Yaskawa INFORM job: R1_W24(-90,90)KM-OK.JBI

/JOB
//NAME R1_W24(-90,90)KM-OK
///FOLDERNAME SCIANA-NOWY-R2-KM
//POS
///NPOS 55,55,0,5,0,0
///TOOL 0
///POSTYPE PULSE
///PULSE
C00000=-125210,-84514,-96282,42678,80589,-84145
C00001=-120727,25071,-5570,41830,73546,-76217
C00002=-120731,25851,-8598,41444,75264,-75512
C00003=-122137,52036,20168,42709,72709,-77203
C00004=-120675,58589,29768,42747,70121,-77648
C00005=-120167,58596,29776,42572,69880,-77517
C00006=-120675,58589,29768,42747,70121,-77648
C00007=-120675,58540,30899,42917,69583,-77884
C00008=-120675,58589,29768,42747,70121,-77648
C00009=-120675,58477,29643,42742,70137,-77641
C00010=-122267,58661,28071,43051,71685,-77708
C00011=-120675,58477,29643,42742,70137,-77641
C00012=-120223,58483,29649,42586,69921,-77523
C00013=-120675,58477,29643,42742,70137,-77641
C00014=-120675,58430,30663,42897,69653,-77855
C00015=-120675,58477,29643,42742,70137,-77641
C00016=-127422,61486,21154,43844,78340,-77144
C00017=-103662,71226,20496,-9632,86815,-77299
C00018=-86138,65266,24877,-44765,91557,-78354
C00019=-89288,46121,11206,-46267,89248,-79163
C00020=-90123,47165,13689,-45982,87906,-79135
C00021=-91284,46293,12750,-45831,87652,-79337
C00022=-90585,47165,13689,-45982,87906,-79135
C00023=-90585,46982,14567,-45988,87456,-78926
C00024=-90585,47165,13689,-45982,87906,-79135
C00025=-86278,47795,10236,-46953,91764,-78966
C00026=-87175,53657,16657,-46727,90663,-78854
C00027=-89651,46102,11966,-46181,88733,-79090
C00028=-89759,44245,10799,-46054,88265,-79150
C00029=-90806,43557,10070,-45936,88060,-79307
C00030=-90254,44245,10799,-46054,88265,-79150
C00031=-90254,44075,11568,-46055,87869,-78967
C00032=-90254,44245,10799,-46054,88265,-79150
C00033=-84762,54495,12176,-47423,94073,-79385
C00034=-101724,51783,-8903,-10262,98728,-75981
C00035=-116477,36058,-18464,22005,90218,-74000
C00036=-120736,36843,4915,41908,73244,-76347
C00037=-121502,36632,5958,42324,73034,-76779
C00038=-125287,25882,-20546,42352,82844,-74334
C00039=-123287,21349,-12248,42448,76368,-76169
C00040=-120314,21476,-8134,41723,73154,-76197
C00041=-120490,59955,31917,42829,69575,-77806
C00042=-120700,58991,30328,42785,70035,-77700
C00043=-122523,66923,35761,43242,71450,-77933
C00044=-120731,36671,5988,42047,72678,-76581
C00045=-105723,54235,-13578,-3991,98004,-77233
C00046=-123048,56423,20709,-36609,73065,-87559
C00047=-124984,57953,26941,-36441,69789,-87236
C00048=-120736,36842,4915,41908,73246,-76345
C00049=-121502,36633,5957,42324,73034,-76779
C00050=-124978,61821,31571,-36625,69095,-86989
C00051=-125030,62392,32007,-36598,69092,-87009
C00052=-121851,45443,10259,-36933,74193,-87458
C00053=-115427,43228,-13903,-33045,78422,-89398
C00054=-52589,-18739,-88829,-40097,82225,-62604
BC00000=161746,674682,1001873
BC00001=160601,672229,1019985
BC00002=160643,672224,912451
BC00003=166290,673398,893644
BC00004=166290,668100,893644
BC00005=166290,668100,893644
BC00006=166290,668100,893644
BC00007=166290,668100,893644
BC00008=166290,668100,893644
BC00009=149811,742558,923347
BC00010=166290,742558,893644
BC00011=166290,742558,893644
BC00012=166290,742558,893644
BC00013=166290,742558,893644
BC00014=166290,742558,893644
BC00015=166290,742558,893644
BC00016=166290,742558,893644
BC00017=166290,742558,893644
BC00018=166290,766679,893644
BC00019=166290,766679,893644
BC00020=166290,766679,893644
BC00021=166290,766679,893644
BC00022=166290,766679,893644
BC00023=166290,766679,893644
BC00024=166290,766679,893644
BC00025=166290,766679,893644
BC00026=166290,702046,893644
BC00027=166290,702046,893644
BC00028=166290,702046,893644
BC00029=166290,702046,893644
BC00030=166290,702046,893644
BC00031=166290,702046,893644
BC00032=166290,702046,893644
BC00033=166290,702046,893644
BC00034=166638,702119,892274
BC00035=166935,702182,891102
///LIMIT ON
BC00036=168548,660891,886121
BC00037=168548,660891,886121
///LIMIT OFF
BC00038=167124,702222,890357
BC00039=167124,702222,890357
BC00040=167124,702222,890357
BC00041=167124,702222,890357
BC00042=168177,754669,886217
BC00043=168295,739818,888985
BC00044=160389,716827,912081
BC00045=168295,689338,885751
BC00046=273959,665226,893644
BC00047=273959,665226,893644
///LIMIT ON
BC00048=168822,599448,886521
BC00049=168822,599448,886521
///LIMIT OFF
BC00050=273959,700483,893644
BC00051=273959,750908,893644
BC00052=273959,756458,893644
BC00053=273959,714241,893644
BC00054=115457,714241,893644
///POSTYPE BASE
///RECTAN
///RCONF 0,0,0,0,0,0,0,0,0,0,0,0,0,0,0,0,0,0,0,0,0,0,0,0
P00006=0.222,-3.123,-1.508,0.0000,0.0000,0.0000
P00021=-0.225,-6.128,-0.405,0.0000,0.0000,0.0000
P00022=0.222,-3.123,-1.508,0.0000,0.0000,0.0000
P00023=0.143,-0.036,0.682,0.0000,0.0000,0.0000
P00024=0.145,-0.552,1.326,0.0000,0.0000,0.0000
//INST
///DATE 2024/07/29 11:47
///ATTR SC,RW
///GROUP1 RB1,BS1
NOP
SFTOF
CALL JOB:CLEAN-R1_KM_NEW_SCIANA
MOVJ C00000 BC00000 VJ=100.00
MOVJ C00001 BC00001 VJ=100.00
MOVJ C00002 BC00002 VJ=100.00
SFTOF
MOVJ C00003 BC00003 VJ=100.00
MOVL C00004 BC00004 V=166.7
REFP 3 C00005 BC00005
CALL JOB:SEARCH-R1
SET P021 P006
SFTON P021
MOVL C00006 BC00006 V=166.7
REFP 3 C00007 BC00007
CALL JOB:SEARCH-R1
SET P021 P006
SFTON P021
MOVL C00008 BC00008 V=166.7
SFTOF
MOVJ C00009 BC00009 VJ=100.00
MOVJ C00010 BC00010 VJ=100.00
MOVL C00011 BC00011 V=166.7
REFP 3 C00012 BC00012
CALL JOB:SEARCH-R1
SET P022 P006
SFTON P022
MOVL C00013 BC00013 V=166.7
REFP 3 C00014 BC00014
CALL JOB:SEARCH-R1
SET P022 P006
SFTON P022
MOVL C00015 BC00015 V=166.7
SFTOF
MOVJ C00016 BC00016 VJ=100.00
MOVJ C00017 BC00017 VJ=30.00
MOVJ C00018 BC00018 VJ=100.00
MOVJ C00019 BC00019 VJ=100.00
MOVL C00020 BC00020 V=166.7
REFP 3 C00021 BC00021
CALL JOB:SEARCH-R1
SET P023 P006
SFTON P023
MOVL C00022 BC00022 V=166.7
REFP 3 C00023 BC00023
CALL JOB:SEARCH-R1
SET P023 P006
SFTON P023
MOVL C00024 BC00024 V=166.7
SFTOF
MOVJ C00025 BC00025 VJ=100.00
MOVJ C00026 BC00026 VJ=100.00
MOVJ C00027 BC00027 VJ=100.00
MOVL C00028 BC00028 V=166.7
REFP 3 C00029 BC00029
CALL JOB:SEARCH-R1
SET P024 P006
SFTON P024
MOVL C00030 BC00030 V=166.7
REFP 3 C00031 BC00031
CALL JOB:SEARCH-R1
SET P024 P006
SFTON P024
MOVL C00032 BC00032 V=166.7
SFTOF
MOVJ C00033 BC00033 VJ=100.00
MOVJ C00034 BC00034 VJ=30.00
MOVJ C00035 BC00035 VJ=100.00
REFP 1 C00036 BC00036
REFP 2 C00037 BC00037
MOVJ C00038 BC00038 VJ=100.00
SFTON P021
MOVJ C00039 BC00039 VJ=100.00
MOVL C00040 BC00040 V=166.7
MACRO1 MJ#(0) ARGF9
ARCON
SFTON P022
MOVL C00041 BC00041 V=9.2
MOVL C00042 BC00042 V=9.2
ARCOF
SFTOF
MOVL C00043 BC00043 V=333.3
MOVL C00044 BC00044 V=500.0
MOVJ C00045 BC00045 VJ=100.00
MOVJ C00046 BC00046 VJ=100.00
SFTON P024
MOVL C00047 BC00047 V=166.7 PL=0
REFP 1 C00048 BC00048
REFP 2 C00049 BC00049
MACRO1 MJ#(0) ARGF9
ARCON
MOVL C00050 BC00050 V=9.2
SFTON P023
MOVL C00051 BC00051 V=9.2
ARCOF
SFTOF
MOVL C00052 BC00052 V=333.3
MOVL C00053 BC00053 V=500.0
MOVJ C00054 BC00054 VJ=100.00
END
